(* CoDeSys 2.3.9.28 project: devicedriver_cooling_v1_0.pro *)
(* Libraries: Standard.lib 10.4.12 16:12:40, lib60.lib 14.4.12 13:00:06, lib60_data_types.lib 10.4.12 16:12:40 *)

(* PLC configuration (modules and I/O channels)
adc_hw_w_pin_0 AT %IW0 [ADC_val] mV/uA/Ohm
adc_hw_w_pin_0_fresh AT %IW2 [Error_Code]
adc_hw_w_pin_1 AT %IW4 [ADC_val] mV/uA/Ohm
adc_hw_w_pin_1_fresh AT %IW6 [Error_Code]
adc_hw_w_pin_2 AT %IW8 [ADC_val] mV/uA/Ohm
adc_hw_w_pin_2_fresh AT %IW10 [Error_Code]
Not used [not_used] node 3, in %IB12 out %QB0
Not used [not_used] node 4, in %IB12 out %QB0
Not used [not_used] node 5, in %IB12 out %QB0
Not used [not_used] node 6, in %IB12 out %QB0
Not used [not_used] node 7, in %IB12 out %QB0
ADC_32V range configured by SW [ADC_Range_by_SW] node 1, in %IB12 out %QB0 {ADC_Range = 0-5V; ADC_Range = 0-5V}
  Not used [not_used] node 0, in %IB12 out %QB0
  Not used [not_used] node 1, in %IB12 out %QB0
  Not used [not_used] node 2, in %IB12 out %QB0
  Not used [not_used] node 3, in %IB12 out %QB0
  Not used [not_used] node 4, in %IB12 out %QB0
  Not used [not_used] node 5, in %IB12 out %QB0
  Not used [not_used] node 6, in %IB12 out %QB0
  Not used [not_used] node 7, in %IB12 out %QB0
PWM Current Measurement or DigOUT [DO_or_PWM_CM] node 2, in %IB12 out %QB0
  Not used [not_used] node 0, in %IB12 out %QB0
  Not used [not_used] node 1, in %IB12 out %QB0
  Not used [not_used] node 2, in %IB12 out %QB0
  Not used [not_used] node 3, in %IB12 out %QB0
TimerIN or AnalogIN or DigitalIN [Timer_IN] node 3, in %IB12 out %QB0
  Not used [not_used] node 0, in %IB12 out %QB0
  Not used [not_used] node 1, in %IB12 out %QB0
  Not used [not_used] node 2, in %IB12 out %QB0
  Not used [not_used] node 3, in %IB12 out %QB0
DigIN [Dig_IN] node 4, in %IB12 out %QB0
  Not used [not_used] node 0, in %IB12 out %QB0
  Not used [not_used] node 1, in %IB12 out %QB0
  Not used [not_used] node 2, in %IB12 out %QB0
  Not used [not_used] node 3, in %IB12 out %QB0
  Not used [not_used] node 4, in %IB12 out %QB0
  Not used [not_used] node 5, in %IB12 out %QB0
  Not used [not_used] node 6, in %IB12 out %QB0
  Not used [not_used] node 7, in %IB12 out %QB0
PWM or TimerIN or DigitalIN or DigOUT [PWM_or_TI_or_DI_or_DO] node 5, in %IB12 out %QB0
  PWM 0 [IO_PWM_00] node 0, in %IB12 out %QB0 {PWM_Frequency = 200; PWM_Polarity = high time variable; PWMCM_Channel = No Current Measurement; PWM_DiagMargin = 250us diagnostic margin}
    PWM_0_duty AT %QW0 [PWM_Duty]
    PWM_0_stat AT %IW12 [Error_Code]
  Not used [not_used] node 1, in %IB14 out %QB2
  Not used [not_used] node 2, in %IB14 out %QB2
  Not used [not_used] node 3, in %IB14 out %QB2
  Not used [not_used] node 4, in %IB14 out %QB2
  Not used [not_used] node 5, in %IB14 out %QB2
  Not used [not_used] node 6, in %IB14 out %QB2
  Not used [not_used] node 7, in %IB14 out %QB2
DigOUT or AnalogIN [DigOUT_or_AnIN] node 6, in %IB14 out %QB2
  Not used [not_used] node 0, in %IB14 out %QB2
  Not used [not_used] node 1, in %IB14 out %QB2
  Not used [not_used] node 2, in %IB14 out %QB2
  Not used [not_used] node 3, in %IB14 out %QB2
  Not used [not_used] node 4, in %IB14 out %QB2
  Not used [not_used] node 5, in %IB14 out %QB2
  Not used [not_used] node 6, in %IB14 out %QB2
  Not used [not_used] node 7, in %IB14 out %QB2
Interfaces [INTERFAC] node 7, in %IB14 out %QB2
  Not used [not_used] node 0, in %IB14 out %QB2
  Not used [not_used] node 1, in %IB14 out %QB2
  Not used [not_used] node 2, in %IB14 out %QB2
  Not used [not_used] node 3, in %IB14 out %QB2
Retain_stat AT %IW14 [Error_Code]
PWM_Enable AT %QB2 [PWM_Enable]
Sleep_Mode AT %QB3 [Sleep_Mode]
K15 AT %IW16 [Dig_IN_val] PIN 271
SS0_val AT %IW18 [ADC_val] mV
SS0_fresh AT %IW20 [Error_Code]
SS1_val AT %IW22 [ADC_val] mV
SS1_fresh AT %IW24 [Error_Code]
SS_var_val AT %IW26 [ADC_val] mV
SS_var_fresh AT %IW28 [Error_Code]
Board_temp_val AT %ID30 [Boardtemp_val] °C
Board_temp_fresh AT %IW34 [Error_Code]
Battery_val AT %IW36 [ADC_val] mV
Battery_fresh AT %IW38 [Error_Code]
CycleLoad AT %ID40 [Time_val] us
CycleLoadMin AT %ID44 [Time_val] us
CycleLoadMax AT %ID48 [Time_val] us
ResetLoadStat AT %QB4 [ResetStats]
*)

(* Task configuration *)
TASK Task_10ms (PRIORITY := 1, INTERVAL := T#50ms);
	cooling();
END_TASK

(* Global variable list: adc_Public *)
VAR_GLOBAL

	adc_inf_r_ntc0_temp: REAL; 	(* Temperature of NTC 0 in °C *)
	adc_inf_r_ntc1_temp: REAL;	(* Temperature of NTC 1 in °C *)
	adc_inf_r_ntc2_temp: REAL;	(* Temperature of NTC 2 in °C *)

END_VAR

(* Global variable list: cooling_Public *)
VAR_GLOBAL

	cooling_ctrl_b_enable: BOOL;			(* Enable all Cooling-Systems *)
	cooling_inf_b_cooling_active: BOOL;		(* Display active cooling State *)
	cooling_inf_b_cooldown_active: BOOL;	(* Display active cooldown State *)

END_VAR

(* Global variable list: gpio_Public *)
VAR_GLOBAL

	gpio_ctrl_b_fan1_value: BOOL;	(* Controlls Fan No. 1*)
	gpio_ctrl_b_pump1_value: BOOL;	(* Controlls Pump No. 1*)

END_VAR

(* POU cooling, ST *)
PROGRAM cooling
VAR

	cooling_state: INT :=0;		(* Statemachine Step Variable *)

	cooling_cooldownTimer: TP;	(* Pulse Generator for cooldown time *)

END_VAR

VAR CONSTANT

	COOLING_COOLDOWNTIME: TIME := T#5s;	(* Minimal cooldown-time *)

	COOLING_MAX_TEMPTERATURE: INT := 35;	(* Temperature where fans start *)
	COOLING_MIN_TEMPTERATURE: INT := 25;	(* Temperature where fans stop *)


END_VAR
(********************************************************************************************************************************************************************
Programm		cooling
Level			Devicedriver
Project			Suncar-Bagger
Autor			Jürg Horisberger
Date			03.04.2014
Version:		1.1
Controlled:		

Changelog:

Version		User/Date		Changes
-------		---------		-------
0.1			jho/30.3.14		Initial version
0.2			jho/1.4.14		Change from FB to PRG, Private variables moved to PRG-Header
0.3			jho/2.4.14		Moved information outputs to Output controll
0.4			jho/2.4.14		Removed Output controll -> All Actions done in the StateMachine, Inserted Substates 21 and 22

1.0			jho/3.4.14		Renamed all Variables according to Document: "UML Statediagramm: Cooling" v
1.1			tzi/12.4.14		testen was github macht mit projekt

		
Description:
	- Controlls Pump and Fan of the cooling-cirquit. 
	- Has a defined cool-down period and continues to run until predefined temperature is reached

Used public variables:

	controll input
		
		cooling_ctrl_b_enable			(* Enable all Cooling-Systems *)

	information output

		cooling_inf_b_cooling_active	(* Display active cooling State *)
		cooling_inf_b_cooldown_active	(* Display active cooldown State *)

	information input
		
		adc_inf_r_ntc0_temp			 	(* Temperature of NTC 0 in °C *)

	controll output
		
		gpio_ctrl_b_fan1_value			(* Controlls Fan No. 1*)
		gpio_ctrl_b_pump1_value			(* Controlls Pump No. 1*)

********************************************************************************************************************************************************************)

(* Set variables for cooldown-timer*)
cooling_cooldownTimer(IN := cooling_inf_b_cooldown_active, PT:= COOLING_COOLDOWNTIME);



(*State Machine: cooling*)
(*======================*)

CASE cooling_state OF

		0:(* Initialize *);
			cooling_inf_b_cooling_active := FALSE;		(*Set all controll outputs to initial State *)
			cooling_inf_b_cooldown_active := FALSE;
			gpio_ctrl_b_pump1_value := FALSE;
			gpio_ctrl_b_fan1_value := FALSE;
			cooling_state:= 1;


		1:(*Idle *)
			IF cooling_ctrl_b_enable THEN			(* If Enable all Cooling-Systems *)
				gpio_ctrl_b_pump1_value := TRUE;
				cooling_inf_b_cooling_active := TRUE;
				cooling_state:= 21;
			END_IF
		21:(*Active-Wait*)
			IF NOT cooling_ctrl_b_enable THEN		(* If Disable all Cooling-Systems *)
				gpio_ctrl_b_fan1_value := TRUE;
				cooling_inf_b_cooling_active := FALSE;
				cooling_inf_b_cooldown_active := TRUE;
				cooling_state:= 3;
			END_IF

			IF (adc_inf_r_ntc0_temp > COOLING_MAX_TEMPTERATURE) THEN	(* If to hot go to "Acitve-fan_active" State*)
				gpio_ctrl_b_fan1_value := TRUE;
				cooling_state:= 22;
			END_IF



IF(adc_inf_r_ntc0_temp < COOLING_MIN_TEMPTERATURE)	THEN	(* If cold enough go to "Active-Wait" State*)
				gpio_ctrl_b_fan1_value := FALSE;
				cooling_state:= 21;
			END_IF

		22:(*Acitve-fan_active*)
			IF NOT cooling_ctrl_b_enable THEN		(* If Disable all Cooling-Systems *)
				cooling_inf_b_cooling_active := FALSE;
				cooling_inf_b_cooldown_active := TRUE;
				cooling_state:= 3;
			END_IF

			IF(adc_inf_r_ntc0_temp < COOLING_MIN_TEMPTERATURE)	THEN	(* If cold enough go to "Active-Wait" State*)
				gpio_ctrl_b_fan1_value := FALSE;
				cooling_state:= 21;
			END_IF


		3:(* Cooldown *)
			IF (NOT cooling_cooldownTimer.Q) AND (adc_inf_r_ntc0_temp < COOLING_MIN_TEMPTERATURE) THEN		(* Wait for cooldown-Timer to expire and temperatures to drop *)
				cooling_inf_b_cooldown_active := FALSE;
				gpio_ctrl_b_pump1_value := FALSE;
				gpio_ctrl_b_fan1_value := FALSE;
				cooling_state:= 1;
			END_IF


END_CASE
END_PROGRAM

(* POU PLC_PRG, ST *)
PROGRAM PLC_PRG
VAR
	nop: BOOL;
END_VAR
nop; (* Do nothing. All Blocks are called as seperate Tasks! *)
END_PROGRAM

(* Visualisation cooling_testbench
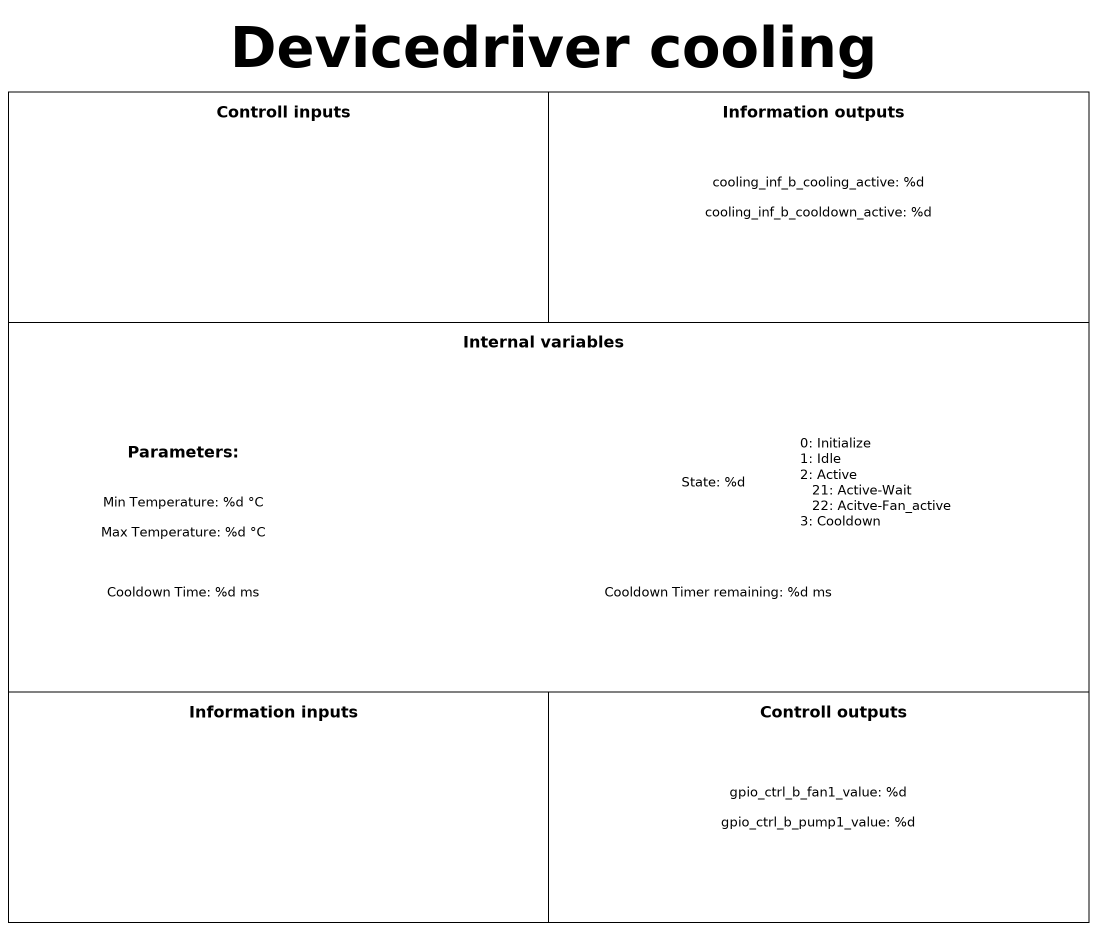
rectangle at (580,160)-(1101,201): text "cooling_inf_b_cooling_active: %d"; shows cooling_inf_b_cooling_active
rectangle at (580,190)-(1101,231): text "cooling_inf_b_cooldown_active: %d"; shows cooling_inf_b_cooldown_active
rectangle at (130,100)-(481,121): text "Controll inputs"
rectangle at (660,100)-(1011,121): text "Information outputs"
rectangle at (120,700)-(471,721): text "Information inputs"
rectangle at (680,700)-(1031,721): text "Controll outputs"
rectangle at (390,330)-(741,351): text "Internal variables"
rectangle at (610,460)-(861,501): text "State: %d"; shows cooling.cooling_state
rectangle at (80,570)-(331,611): text "Cooldown Time: %d ms"; shows cooling.cooling_cooldowntime
rectangle at (600,570)-(881,611): text "Cooldown Timer remaining: %d ms"; shows cooling.cooling_cooldowntime - cooling.cooling_cooldowntimer.ET
rectangle at (80,480)-(331,521): text "Min Temperature: %d °C"; shows cooling.COOLING_MIN_TEMPTERATURE
rectangle at (80,510)-(331,551): text "Max Temperature: %d °C"; shows cooling.COOLING_MAX_TEMPTERATURE
rectangle at (30,440)-(381,461): text "Parameters:"
rectangle at (580,770)-(1101,811): text "gpio_ctrl_b_fan1_value: %d"; shows gpio_ctrl_b_fan1_value
rectangle at (580,800)-(1101,841): text "gpio_ctrl_b_pump1_value: %d"; shows gpio_ctrl_b_pump1_value
rectangle at (820,410)-(1011,551): text "0: Initialize / 1: Idle / 2: Active / 21: Active-Wait / 22: Acitve-Fan_active / 3: Cooldown"
rectangle at (230,0)-(921,91): text "Devicedriver cooling"
5 more shapes without text or variables
2 elements of other kinds (tables, trends, ...) not read
*)

(* Visualisation VCU_Stats
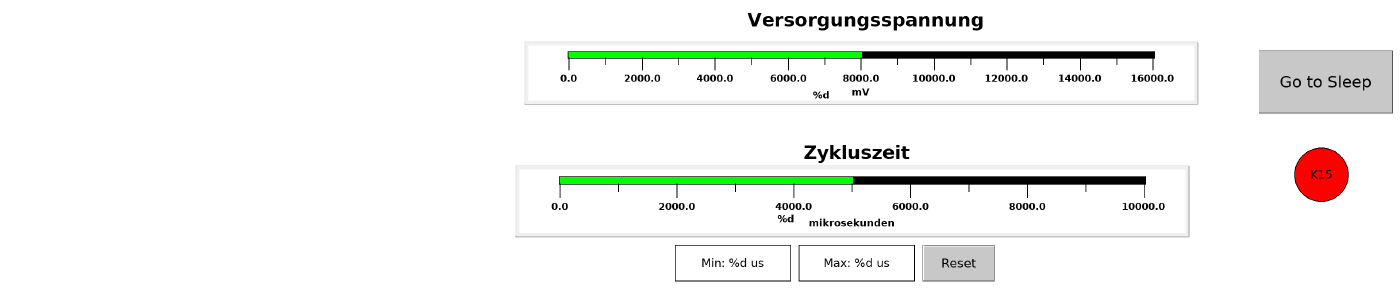
ellipse at (970,230)-(1031,291): text "K15"; alarm colour if K15
group at (90,250)-(851,331)
  rectangle at (0,0)-(1,1): text "{ExtendedElement},Visu\ElementDLL.ete,1,@Bargraph,761,71,0,0,0,CycleLoad,mikrosekunden,%.1f,1000,2000,0,10000,0,0,0,0,0,0,0,-13,16,700,Arial,0,255,0,255,0,0,0,0,1,1,0,0,0,,0,0,0,"
  rectangle at (50,12)-(381,18): alarm colour if (CycleLoad) < 0; right ((CycleLoad * 1.0) - 5000)  * 0.066
  rectangle at (38,34)-(62,66): text "0.0"
  rectangle at (156,34)-(208,66): text "2000.0"
  rectangle at (288,34)-(340,66): text "4000.0"
  rectangle at (420,34)-(472,66): text "6000.0"
  rectangle at (552,34)-(604,66): text "8000.0"
  rectangle at (679,34)-(740,66): text "10000.0"
  rectangle at (283,49)-(477,65): text "mikrosekunden"
rectangle at (330,220)-(621,251): text "Zykluszeit"
group at (100,110)-(861,181)
  rectangle at (0,0)-(1,1): text "{ExtendedElement},Visu\ElementDLL.ete,1,@Bargraph,761,71,0,0,0,Battery_val,mV,%.1f,1000,2000,0,16000,0,0,0,0,0,0,0,-13,16,700,Arial,0,255,0,255,0,0,0,0,1,1,0,0,0,,0,0,0,"
  rectangle at (50,12)-(381,18): alarm colour if (Battery_val) < 0; right ((Battery_val * 1.0) - 8000)  * 0.04125
  rectangle at (38,34)-(62,66): text "0.0"
  rectangle at (107,34)-(159,66): text "2000.0"
  rectangle at (189,34)-(241,66): text "4000.0"
  rectangle at (272,34)-(324,66): text "6000.0"
  rectangle at (354,34)-(406,66): text "8000.0"
  rectangle at (432,34)-(493,66): text "10000.0"
  rectangle at (514,34)-(575,66): text "12000.0"
  rectangle at (597,34)-(658,66): text "14000.0"
  rectangle at (679,34)-(740,66): text "16000.0"
  rectangle at (359,49)-(401,65): text "mV"
rectangle at (340,70)-(631,101): text "Versorgungsspannung"
button at (930,120)-(1081,191): text "Go to Sleep"; taps Sleep_Mode
rectangle at (370,300)-(421,321): text "%d"; shows CycleLoad
rectangle at (410,160)-(461,181): text "%d"; shows Battery_val
rectangle at (270,340)-(401,381): text "Min: %d us"; shows CycleLoadMin
rectangle at (410,340)-(541,381): text "Max: %d us"; shows CycleLoadMax
button at (550,340)-(631,381): text "Reset"; taps ResetLoadStat
46 more shapes without text or variables
*)
